KUKA KRL program: C3_getcube.src, C3_getcube.dat

--- C3_getcube.src ---
&ACCESS RVO
&REL 4
&PARAM DISKPATH = KRC:\R1\Program
DEF C3_getcube (COORD:IN)

DECL FRAME COORD

;FOLD INI;%{PE}
  ;FOLD BASISTECH INI
    GLOBAL INTERRUPT DECL 3 WHEN $STOPMESS==TRUE DO IR_STOPM ( )
    INTERRUPT ON 3
    BAS (#INITMOV,0 )
  ;ENDFOLD (BASISTECH INI)
  ;FOLD USER INI
    ;Make your modifications here

  ;ENDFOLD (USER INI)
;ENDFOLD (INI)

;FOLD PTP HOME  Vel= 100 % DEFAULT;%{PE}%MKUKATPBASIS,%CMOVE,%VPTP,%P 1:PTP, 2:HOME, 3:, 5:100, 7:DEFAULT
;$BWDSTART = FALSE
;PDAT_ACT=PDEFAULT
;FDAT_ACT=FHOME
;BAS (#PTP_PARAMS,100 )
;$H_POS=XHOME
;PTP  XHOME
;ENDFOLD

; Fahre Coord an
      $BASE = base_data[6]
      $TOOL = tool_data[14]

      GRPg_SetStateAndCheck(1, 1, 0.2, 1)

      COORD.Z = COORD.Z - 60

      ;Fahre Pos mit Z + 30 an
      SPTP COORD

      ;Senke auf Plazierpos
      COORD.Z = COORD.Z + 60
      SLIN COORD

      ;Platziere
      GRPg_SetStateAndCheck(1, 2, 0.2, 0)

      ;Hebe auf Pos mit Z + 30
      COORD.Z = COORD.Z - 60
      SLIN COORD



;FOLD PTP HOME  Vel= 100 % DEFAULT;%{PE}%MKUKATPBASIS,%CMOVE,%VPTP,%P 1:PTP, 2:HOME, 3:, 5:100, 7:DEFAULT
;$BWDSTART = FALSE
;PDAT_ACT=PDEFAULT
;FDAT_ACT=FHOME
;BAS (#PTP_PARAMS,100 )
;$H_POS=XHOME
;PTP  XHOME
;ENDFOLD

END

--- C3_getcube.dat ---
&ACCESS RVO
&REL 4
&PARAM DISKPATH = KRC:\R1\Program
DEFDAT  C3_getcube PUBLIC

DECL E6POS XP1={X 224.960861,Y 55.9276581,Z 35.7754402,A 162.906586,B 89.0492325,C -106.826286,S 2,T 10,E1 0.0,E2 0.0,E3 0.0,E4 0.0,E5 0.0,E6 0.0}
DECL FDAT FP1={TOOL_NO 14,BASE_NO 2,IPO_FRAME #BASE,POINT2[] " ",TQ_STATE FALSE}
DECL PDAT PPDAT1={VEL 100.000,ACC 100.000,APO_DIST 100.000,GEAR_JERK 50.0000,EXAX_IGN 0}


ENDDAT
